TYPE MOTION_LOGGER_MSG : STRING(128); END_TYPE

(* stored: Version 1.1.0.1
   DUT MOTION_LOGGER_MSG: Id {a5f6d85b-a42a-48cd-968a-055b69703b65} *)
